// TIA Portal V19 export
TYPE "C402_STU_VKL_TYPIC"
   STRUCT
      CMD { ExternalAccessible := 'False'; ExternalVisible := 'False'; ExternalWritable := 'False'} : USInt;   // Sturing verkeerslicht
      CMD_ONHD { ExternalAccessible := 'False'; ExternalVisible := 'False'; ExternalWritable := 'False'} : USInt;   // Automatische onderhoudstesten uitvoeren
      SNEL { ExternalAccessible := 'False'; ExternalVisible := 'False'; ExternalWritable := 'False'} : USInt;   // Sturing versneld
   END_STRUCT;
END_TYPE
